PROGRAM P_FehlerAllgemein
VAR
	fbKontrolleEndschalter : FB_KontrolleEndschalter;
END_VAR

(* Baustein: FC3 Fehlererkennung allgemein *)
(* Name: FEHL_ERK *)
(* Zeitstempel Code: 19.10.2011 10:02:13 *)
(* Interface: 09.07.2010 10:27:01 *)

F_KontrollZeiten();

F_Doppelmeldung(); //OK

F_AusloeseschalterDauermeldung(); //noch ohne Wirkung

fbKontrolleEndschalter(errorOffset := 600); //OK - 600er ID-Bereich

//F_Aufstarten();

F_FehlerAufgetreten();
(*
IF F_FehlerAufgetreten() THEN
	F_StoerungsbitsAuswerten();
END_IF
*)

END_PROGRAM

(* stored: Version 1.1.0.1, ProductVersion 3.1.4024.3
   POU P_FehlerAllgemein: Id {82b7a904-a1be-42ee-894f-6421b6623774}, SpecialFunc None *)
